INTERFACE InterfaceContainer EXTENDS __SYSTEM.IQueryInterface

PROPERTY active_futures : UINT
GET
END_GET
END_PROPERTY

PROPERTY num_of_future : UINT
GET
END_GET
END_PROPERTY

METHOD reset_sub_futures : BOOL
VAR_INPUT
END_VAR
END_METHOD

END_INTERFACE

(* stored: Version 1.1.0.1, ProductVersion 3.1.4024.12
   Itf InterfaceContainer: Id {24bfec70-0f3a-4ec1-a89e-5407d9c94d6d}
   Property active_futures: Id {2d416ece-2dc1-4b01-a1fe-d0b196d80eaa}
   Get Get: Id {9f74c5c8-3fa8-4c0a-9b16-6bb5d20b0f71}
   Property num_of_future: Id {f8eb50f2-28cd-44d4-9501-560037cfcc71}
   Get Get: Id {9e329e0b-c0dd-4e74-8ae7-beef2f01ea63}
   Method reset_sub_futures: Id {2b4aedc3-0b4d-4f4c-b2aa-df9f403a1db1} *)
